{attribute 'qualified_only'}
VAR_GLOBAL
	
	// Barra Posicionamiento Bases
	{attribute 'OPC.UA.DA' := '1'}
	cerrarAbrazaderaBase : BOOL;
	{attribute 'OPC.UA.DA' := '1'}
	levantarAbrazaderaBase : BOOL;
	{attribute 'OPC.UA.DA' := '1'}
	limiteSujeccionBase : BOOL;
	{attribute 'OPC.UA.DA' := '1'}
	limiteVerticalBase : BOOL;
	
	// Barra posicionamiento Tapas
 	{attribute 'OPC.UA.DA' := '1'}
	levantarAbrazaderaTapa : BOOL;
	{attribute 'OPC.UA.DA' := '1'}
	cerrarAbrazaderaTapa : BOOL;
	{attribute 'OPC.UA.DA' := '1'}
	limiteSujeccionTapa : BOOL;
	{attribute 'OPC.UA.DA' := '1'}
	limiteVerticalTapa : BOOL;
 
	// SENSORES
	{attribute 'OPC.UA.DA' := '1'}
	sensorFotoBase : BOOL;;
	{attribute 'OPC.UA.DA' := '1'}
	sensorFotoTapa : BOOL;
	{attribute 'OPC.UA.DA' := '1'}
	sensorPostSellado : BOOL;
	{attribute 'OPC.UA.DA' := '1'}
	modoManual : BOOL; // Estado 0 del selector
	{attribute 'OPC.UA.DA' := '1'}
	modoAuto : BOOL; // Estado 1 del selector

	
	// Pick & Place

	{attribute 'OPC.UA.DA' := '1'}
	PickPlace_MoverX : BOOL;
	{attribute 'OPC.UA.DA' := '1'}
	PickPlace_MoverZ : BOOL;
	{attribute 'OPC.UA.DA' := '1'}
	PickPlace_Agarrar : BOOL;
	{attribute 'OPC.UA.DA' := '1'}
	PickPlace_Detectado : BOOL;
	{attribute 'OPC.UA.DA' := '1'}
	PickPlace_MovingXY: BOOL;
	{attribute 'OPC.UA.DA' := '1'}
	PickPlace_MovingZ: bool; 
	
	
	// CINTAS
	{attribute 'OPC.UA.DA' := '1'}
	cintaBases : BOOL;
	{attribute 'OPC.UA.DA' := '1'}
	cintaTapas : BOOL;
	
	// CUADRO
	{attribute 'OPC.UA.DA' := '1'}
	 botonStart : BOOL;
	{attribute 'OPC.UA.DA' := '1'}
	 botonStop : BOOL;	
	 {attribute 'OPC.UA.DA' := '1'}
	 botonReset : BOOL;
	{attribute 'OPC.UA.DA' := '1'}
	 luzVerticalVerde : BOOL;
	{attribute 'OPC.UA.DA' := '1'}
	 luzVerticalNaranja : BOOL;
	{attribute 'OPC.UA.DA' := '1'}
	 luzVerticalRoja : BOOL;	
	{attribute 'OPC.UA.DA' := '1'}
	 luzStop : BOOL;  // luz de boton stop
	 {attribute 'OPC.UA.DA' := '1'}
	 luzStart : BOOL; // luz del boton de start
	 {attribute 'OPC.UA.DA' := '1'}
	 luzReset : BOOL; 
	 {attribute 'OPC.UA.DA' := '1'}
	 seta : BOOL; // Seta de emergencia
 

 
END_VAR

(* stored: Version 1.1.0.1, ProductVersion 3.1.4024.15
   GVL GVLvars: Id {b38c3178-7f30-4b50-90fb-76531ebc4cba} *)
